RoboDK station: RoboDK sw04 UR3e mit Robotiq First Test Hindernis.rdk

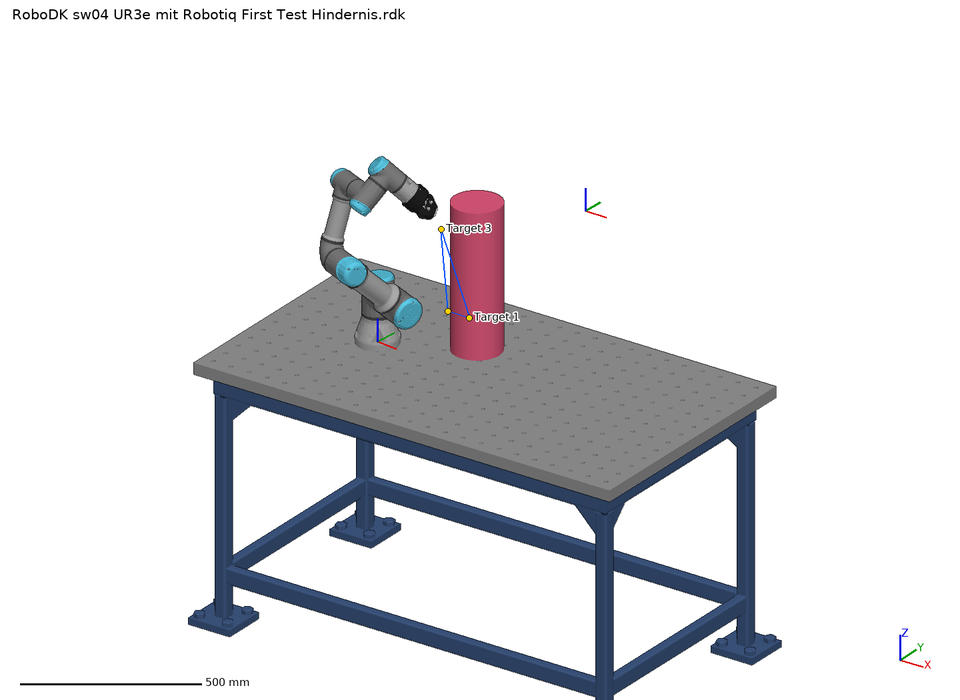
[picture v0: the station drawn from its stored meshes, robots at their saved joint values, targets as dots, program paths as lines]
Station UR3e mit Robotiq First Test Hindernis (saved by RoboDK 5.9.5). Poses are relative to the parent item; angles as X-Y-Z fixed-axis rotations.
Station parameters (name, value as stored): OPC-UA, opc.tcp://localhost:4840
  - frame UR3e Base at (0, 0, 0) mm, rotated rx 0 ry 0 rz -6.26 deg
    - robot UR3e: 6 axes, payload 3 kg, reach 500 mm, repeatability 0.03 mm, weight 11 kg
        modified DH rows (alpha deg, a mm, theta deg, d mm): 0, 0, 0, 151.9; 90, 0, 180, 0; 0, 243.55, 0, 0; 0, 213.2, 0, 131.05; -90, 0, 0, 85.35; 90, 0, 180, 92.1
        joint limits [-360, -360, -360, -360, -360, -360] to [360, 360, 360, 360, 360, 360]; home [0, -90, -90, 0, 90, 0]; saved at [72.664, -43.845, -62.806, -120.838, 68.9, 46.357]
      - robot RobotiQ 2F-85 Gripper (Mechanism) (model RobotiQ 2F85): 1 axes, payload 5 kg
          joint limits [0] to [85]; home [85]; saved at [85]
        - tool Tool 1, TCP at (0, 0, 160) mm
  - object Table 1400x800x800mm at (0, 0, 0) mm, size 1420 x 820 x 800 mm, geometry from Table-1400x800x800mm.sld
    - object Cylinder 150x450mm at (250, 120, 0) mm, size 150 x 150 x 450 mm, geometry from Cylinder-150x450mm.sld
  - frame RobotiQ 2F-85 Gripper (Mechanism) Base at (0, 1000, 0) mm
    - target Target 1 (Cartesian target) at (400.51, -1131.05, 236.31) mm, rotated rx 108.04 ry 86.9 rz -161.94 deg; joints [140.535, 13.829, -29.849, -165.318, 45.782, 93.881] of UR3e
    - target Target 3 (Cartesian target) at (305.3, -1131.05, 480.8) mm, rotated rx -90 ry 0 rz -90 deg; joints [0, -90, -90, 0, 90, 0] of UR3e
    - target Target 2 (Cartesian target) at (329.51, -1131.05, 236.31) mm, rotated rx 177.05 ry 1.7 rz -90.09 deg; joints [5.792, -100.67, -95.278, -77.012, 91.677, -0.468] of UR3e
  - program UR3e_AutoProg (7 instructions, listed below)
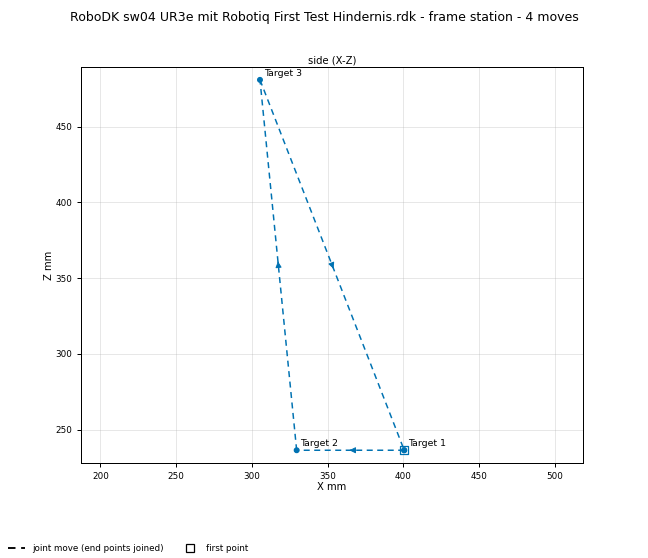
[picture p0: tool path of RoboDK sw04 UR3e mit Robotiq First Test Hindernis.rdk in frame station, 4 of 4 moves have a stored position in this frame; points joined in program order, loops and branches not executed]

--- program UR3e_AutoProg (robot UR3e) ---
  MoveJ (Target 1)
  MoveJ (Target 2)
  Pause 2.0 s
  MoveJ (Target 3)
  Pause 2.0 s
  Pause 2.0 s
  MoveJ (Target 1)
